FUNCTION_BLOCK L1_stul_LD
VAR_INPUT
	CO1: BOOL;
	C5DPR: BOOL;
	C4DPR: BOOL;
END_VAR
VAR_OUTPUT
	MO: BOOL;
	M5DPR: BOOL;
	M4DPR: BOOL;
END_VAR
VAR
END_VAR

// NETWORK 1

END_FUNCTION_BLOCK

(* stored: Version 1.1.0.1, ProductVersion 3.1.4024.13
   POU L1_stul_LD: Id {5c3811d3-69a4-4ae7-81e2-644761434776}, SpecialFunc None *)
